(* PLC project Blank Project, Blank Blank 1.0 *)
(* stored: creationDateTime 2016-05-18T21:14:07, modificationDateTime 2017-02-08T11:15:27 *)

PROGRAM My_Program
  VAR
    var1 AT %IW0.0 : INT := 0;
    var2 AT %IW0.1 : INT := 0;
    var3 AT %IW0.2 : INT := 0;
    var4 AT %QW0.0 : INT;
  END_VAR

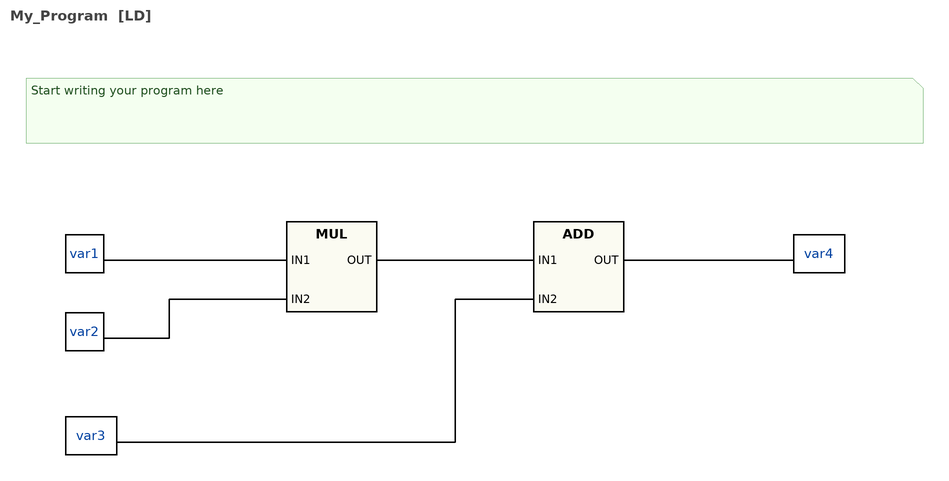
(* LD diagram, written out as Structured Text *)
(* Start writing your program here *)
var4 := var1 * var2 + var3;
END_PROGRAM

CONFIGURATION STD_CONF
  RESOURCE STD_RESSOURCE ON PLC
    TASK TaskMain(INTERVAL := T#50ms, PRIORITY := 0);
    PROGRAM Inst0 WITH TaskMain : My_Program;
  END_RESOURCE
END_CONFIGURATION
